{attribute 'no_assign'}
{attribute 'enable_dynamic_creation'}
{attribute 'no_explicit_call' := 'do not call this POU directly'}
FUNCTION_BLOCK FB_StringBuilder IMPLEMENTS I_StringBuilder, I_Enumerable
VAR CONSTANT
	Default_Capacity : T_Size := 256;
END_VAR
VAR
	{attribute 'hide'} 
	_Capacity : T_Size := THIS^.Default_Capacity;
	{attribute 'hide'} 
	_Length : T_Size := 0;
	_pBuffer : POINTER TO STRING := THIS^.Malloc(THIS^.Capacity);
END_VAR
VAR CONSTANT
	{attribute 'hide'} 
	_fbFree : FB_Free(THIS^._pBuffer) := ();
END_VAR

// Appends the given string to the end of the string builder's contents.
METHOD Append : I_StringBuilder
VAR_INPUT
	sValue : T_LongString;
END_VAR
Append := THIS^.AppendAny(sValue);
END_METHOD

// Appends the given value to the end of the string builder's contents.
METHOD AppendAny : I_StringBuilder
VAR_INPUT
	Value : ANY;
END_VAR
VAR
	bMalloced : BOOL := TRUE;
	Str_Len : T_Size;
	pValue : POINTER TO STRING;
END_VAR
AppendAny := THIS^;
CASE Value.TypeClass OF
	__SYSTEM.TYPE_CLASS.TYPE_STRING: 
		Str_Len := F_StrLen(Value.pValue);
		pValue := Value.pValue;
		bMalloced := FALSE;
		
	__SYSTEM.TYPE_CLASS.TYPE_WSTRING:
		Str_Len := TO_DINT(Tc2_Utilities.WLEN2(Value.pValue));
		pValue := THIS^.Malloc(Str_Len);
		Tc2_Utilities.WSTRING_TO_STRING2(pValue, Value.pValue, TO_UDINT(Str_Len));
		
	__SYSTEM.TYPE_CLASS.TYPE_BOOL,
	__SYSTEM.TYPE_CLASS.TYPE_BYTE,
	__SYSTEM.TYPE_CLASS.TYPE_WORD,
	__SYSTEM.TYPE_CLASS.TYPE_DWORD,
	__SYSTEM.TYPE_CLASS.TYPE_LWORD,
	__SYSTEM.TYPE_CLASS.TYPE_SINT,
	__SYSTEM.TYPE_CLASS.TYPE_INT,
	__SYSTEM.TYPE_CLASS.TYPE_DINT,
	__SYSTEM.TYPE_CLASS.TYPE_LINT,
	__SYSTEM.TYPE_CLASS.TYPE_USINT,
	__SYSTEM.TYPE_CLASS.TYPE_UINT,
	__SYSTEM.TYPE_CLASS.TYPE_UDINT,
	__SYSTEM.TYPE_CLASS.TYPE_ULINT,
	__SYSTEM.TYPE_CLASS.TYPE_REAL,
	__SYSTEM.TYPE_CLASS.TYPE_LREAL,
	__SYSTEM.TYPE_CLASS.TYPE_TIME,
	__SYSTEM.TYPE_CLASS.TYPE_LTIME,
	__SYSTEM.TYPE_CLASS.TYPE_DATE,
	__SYSTEM.TYPE_CLASS.TYPE_DATEANDTIME,
	__SYSTEM.TYPE_CLASS.TYPE_TIMEOFDAY,
	__SYSTEM.TYPE_CLASS.TYPE_POINTER:
		pValue := THIS^.Malloc(SIZEOF(T_LongString));
		pValue^ := F_AnyToString(Value);
		Str_Len := F_StrLen(pValue);
ELSE
	RETURN;
END_CASE

IF (THIS^.Length + Str_Len) >= THIS^.Capacity THEN
	THIS^.Reserve((THIS^.Length + Str_Len + 1)*2);
	END_IF

THIS^.Length := THIS^.Length + Str_Len;
F_StrLCat(THIS^._pBuffer, pValue, THIS^.Length + 1);

IF bMalloced THEN __DELETE(pValue); END_IF
END_METHOD

// !!!UNSAFE!!! THIS WILL APPEND UP TO THE NULL CHARACTER. IF NO NULL EXISTS, THIS WILL RUN FOREVER!
// | Append raw values directly to the internal string buffer. This is meant for appending dynamic strings to the string builder.
METHOD AppendBuffer : I_StringBuilder
VAR_INPUT
	pBuffer : POINTER TO BYTE;
END_VAR
VAR
	Str_Len : T_Size;
END_VAR
AppendBuffer := THIS^;
IF pBuffer = 0 THEN RETURN; END_IF
Str_Len := F_StrLen(pBuffer);

IF (THIS^.Length + Str_Len) >= THIS^.Capacity THEN
	THIS^.Reserve((THIS^.Length + Str_Len + 1)*2);
	END_IF
	
THIS^.Length := THIS^.Length + Str_Len;
F_StrLCat(THIS^._pBuffer, pBuffer, THIS^.Length + 1);
END_METHOD

// Appends a new line (\r\n or $r$n) to string builder's contents.
METHOD AppendLine : I_StringBuilder
AppendLine := THIS^;
THIS^.Append('$r$n');
END_METHOD

// Removes all ASCII white space (spaces, tabs, carriage returns, and linefeeds) from the beginning and end of string in the string builder
METHOD BTrim : I_StringBuilder
VAR
	Start, End, Length : T_Size := 0;
END_VAR
BTrim := THIS^;
IF THIS^.Length = 0 THEN RETURN; END_IF
End := THIS^.Length - 1;

WHILE ((Start <= End) AND THIS^.Is_Space(THIS^._pBuffer^[Start])) DO Start := Start  + 1; END_WHILE
WHILE ((End >= Start) AND THIS^.Is_Space(THIS^._pBuffer^[End])) DO End := End  - 1; END_WHILE

Length := end - start + 1;
F_MemMove(THIS^._pBuffer, ADR(THIS^._pBuffer^[Start]), Length);
THIS^.Length := Length;
THIS^._pBuffer^[THIS^.Length] := 0;
END_METHOD

// Number of bytes allocated in memory for the string builder's contents.
PROPERTY Capacity : T_Size
GET
Capacity := THIS^._Capacity;
END_GET
SET // PROTECTED
THIS^._Capacity := Capacity;
END_SET
END_PROPERTY

// Empties the string builder's contents, resetting its length to zero.
METHOD Clear : I_StringBuilder
Clear := THIS^;
THIS^.Free();
THIS^.Capacity := THIS^.Default_Capacity;
THIS^.Length := 0;
THIS^._pBuffer := THIS^.Malloc(THIS^.Capacity);
THIS^._pBuffer^[0] := 0;
END_METHOD

// Copies a subset of characters in the string builder from specified position at specified length to a string
METHOD CopySubstringTo : I_StringBuilder
VAR_INPUT
	Position, Length : T_Size;
	Value : ANY;
END_VAR
VAR
	pTemp : POINTER TO BYTE;
	pwsTemp : POINTER TO WSTRING;
END_VAR
CopySubstringTo := THIS^;
IF Value.pValue = 0 THEN RETURN; END_IF
CASE Value.TypeClass OF
	__SYSTEM.TYPE_CLASS.TYPE_STRING:
		Length := MIN(Length, Value.diSize - 1);
		IF (Position > THIS^.Length) OR_ELSE (Length <= 0) OR_ELSE (THIS^.Length = 0) THEN Value.pValue[0] := 0; RETURN; END_IF
		F_StrLCpy(Value.pValue, ADR(THIS^._pBuffer^[Position]), Length + 1);
		
	__SYSTEM.TYPE_CLASS.TYPE_WSTRING:
		Length := MIN(Length, (Value.diSize/2) - 1 );
		IF (Position > THIS^.Length) OR_ELSE (Length = 0) OR_ELSE (THIS^.Length = 0) THEN pwsTemp := Value.pValue; pwsTemp^ := ""; RETURN; END_IF
		pTemp := THIS^.Malloc(Length + 1);
		F_StrLCpy(pTemp, ADR(THIS^._pBuffer^[Position]), Length + 1);
		Tc2_Utilities.STRING_TO_WSTRING2(Value.pValue, pTemp, TO_UDINT((Length*2)+1));
		__DELETE(pTemp);
ELSE
	F_StrToAny(Value, THIS^.GetSubstring(Position, Length));
END_CASE
END_METHOD

// Copies contents of string builder to given string of any size
METHOD CopyTo : I_StringBuilder
VAR_INPUT
	Value : ANY;
END_VAR
CopyTo := THIS^;
IF THIS^._pBuffer = 0 THEN Value.pValue[0] := 0; RETURN; END_IF 
CASE Value.TypeClass OF
	__SYSTEM.TYPE_CLASS.TYPE_STRING:
		F_StrLCpy(Value.pValue, THIS^._pBuffer, Value.diSize);
	__SYSTEM.TYPE_CLASS.TYPE_WSTRING:
		Tc2_Utilities.STRING_TO_WSTRING2(Value.pValue, THIS^._pBuffer, TO_UDINT(Value.diSize));
ELSE
	F_StrToAny(Value, THIS^.GetString());
END_CASE
END_METHOD

// Dealloocates String from memory
METHOD PROTECTED Free
VAR_INPUT
END_VAR
IF THIS^._pBuffer <> 0 THEN __DELETE(THIS^._pBuffer); END_IF
THIS^.Capacity := 0;
END_METHOD

// !!!UNSAFE!!! DON'T FORGET TO RELEASE/DELETE FROM	MEMORY WHEN DONE!
// | Get a copy of the internal string buffer at the size of the string length + 1.
METHOD GetBuffer : I_StringBuilder
VAR_IN_OUT
	pBuffer : POINTER TO BYTE;
END_VAR
GetBuffer := THIS^;
pBuffer := THIS^.Malloc(THIS^.Length + 1);
F_StrLCpy(pBuffer, THIS^._pBuffer, THIS^.Length + 1);
END_METHOD

// Retrieves the number of bytes allocated in memory for the string builder's contents.
METHOD GetCapacity : I_StringBuilder
VAR_OUTPUT
	Capacity : T_Size;
END_VAR
GetCapacity := THIS^;
Capacity := THIS^.Capacity;
END_METHOD

// Gets character at specified position in the string builder
METHOD GetChar : T_Char
VAR_INPUT
	Position : T_Size;
END_VAR
IF Position < 0 THEN RETURN; END_IF
IF Position > THIS^.Length THEN RETURN; END_IF
GetChar[0] := THIS^._pBuffer^[Position];
END_METHOD

METHOD GetEnumerator : I_Enumerator
VAR_INST
	fbEnumerator : FB_StringBuilderEnumerator(THIS^);
END_VAR
GetEnumerator := fbEnumerator;
END_METHOD

// Retrieves the current size of string builder contents
METHOD GetLength : I_StringBuilder
VAR_OUTPUT
	Length : T_Size;
END_VAR
GetLength := THIS^;
Length := THIS^.Length;
END_METHOD

// Converts contents of string builder to string and returns them
METHOD GetString : T_LongString
THIS^.CopyTo(GetString);
END_METHOD

// Get a subset of characters in the string builder from specified position at specified length and returns them as a string
METHOD GetSubstring : T_LongString
VAR_INPUT
	Position, Length : T_Size;
END_VAR
THIS^.CopySubstringTo(Position, Length, GetSubstring);
END_METHOD

// Inserts the given string at the specified position.
METHOD Insert : I_StringBuilder
VAR_INPUT
	Position : T_Size;
	sValue : T_LongString;
END_VAR
Insert := THIS^.InsertAny(Position, sValue);
END_METHOD

// Inserts the given value at the specified position.
METHOD InsertAny : I_StringBuilder
VAR_INPUT
	Position : T_Size;
	Value : ANY;
END_VAR
VAR
	bMalloced : BOOL := TRUE;
	Str_Len : T_Size;
	pValue : POINTER TO STRING;
END_VAR
InsertAny := THIS^;
IF Position < 0 OR Position > THIS^.Length THEN RETURN; END_IF 
CASE Value.TypeClass OF
	__SYSTEM.TYPE_CLASS.TYPE_STRING: 
		Str_Len := F_StrLen(Value.pValue);
		pValue := Value.pValue;
		bMalloced := FALSE;
	
	__SYSTEM.TYPE_CLASS.TYPE_WSTRING:
		Str_Len := TO_DINT(Tc2_Utilities.WLEN2(Value.pValue));
		pValue := THIS^.Malloc(Str_Len);
		Tc2_Utilities.WSTRING_TO_STRING2(pValue, Value.pValue, TO_UDINT(Str_Len));

	__SYSTEM.TYPE_CLASS.TYPE_BOOL,
	__SYSTEM.TYPE_CLASS.TYPE_BYTE,
	__SYSTEM.TYPE_CLASS.TYPE_WORD,
	__SYSTEM.TYPE_CLASS.TYPE_DWORD,
	__SYSTEM.TYPE_CLASS.TYPE_LWORD,
	__SYSTEM.TYPE_CLASS.TYPE_SINT,
	__SYSTEM.TYPE_CLASS.TYPE_INT,
	__SYSTEM.TYPE_CLASS.TYPE_DINT,
	__SYSTEM.TYPE_CLASS.TYPE_LINT,
	__SYSTEM.TYPE_CLASS.TYPE_USINT,
	__SYSTEM.TYPE_CLASS.TYPE_UINT,
	__SYSTEM.TYPE_CLASS.TYPE_UDINT,
	__SYSTEM.TYPE_CLASS.TYPE_ULINT,
	__SYSTEM.TYPE_CLASS.TYPE_REAL,
	__SYSTEM.TYPE_CLASS.TYPE_LREAL,
	__SYSTEM.TYPE_CLASS.TYPE_TIME,
	__SYSTEM.TYPE_CLASS.TYPE_LTIME,
	__SYSTEM.TYPE_CLASS.TYPE_DATE,
	__SYSTEM.TYPE_CLASS.TYPE_DATEANDTIME,
	__SYSTEM.TYPE_CLASS.TYPE_TIMEOFDAY,
	__SYSTEM.TYPE_CLASS.TYPE_POINTER:
		pValue := THIS^.Malloc(SIZEOF(T_LongString));
		pValue^ := F_AnyToString(Value);
		Str_Len := F_StrLen(pValue);
ELSE
	RETURN;
END_CASE

IF (THIS^.Length + Str_Len) >= THIS^.Capacity THEN
	THIS^.Reserve((THIS^.Length + Str_Len + 1)*2);
	END_IF

F_MemMove(THIS^._pBuffer + TO_UDINT(Position) + TO_UDINT(Str_Len), THIS^._pBuffer + TO_UDINT(Position), THIS^.Length - Position + 1);
F_MemCpy(THIS^._pBuffer + TO_UDINT(Position), pValue, Str_Len); 
THIS^.Length := THIS^.Length + Str_Len;

IF bMalloced THEN __DELETE(pValue); END_IF
END_METHOD

// !!!UNSAFE!!! THIS WILL INSERT UP TO THE NULL CHARACTER. IF NO NULL EXISTS, THIS WILL RUN FOREVER!
// | Inserts raw values directly to the internal string buffer at the specified position. This is meant for inserting dynamic strings to the string builder.
METHOD InsertBuffer : I_StringBuilder
VAR_INPUT
	Position : T_Size;
	pBuffer : POINTER TO BYTE;
END_VAR
VAR
	Str_Len : T_Size;
END_VAR
InsertBuffer := THIS^;
IF pBuffer = 0 OR Position < 0 OR Position > THIS^.Length THEN RETURN; END_IF
Str_Len := F_StrLen(pBuffer);

IF (THIS^.Length + Str_Len) >= THIS^.Capacity THEN
	THIS^.Reserve((THIS^.Length + Str_Len + 1)*2);
	END_IF

F_MemMove(THIS^._pBuffer + TO_UDINT(Position) + TO_UDINT(Str_Len), THIS^._pBuffer + TO_UDINT(Position), THIS^.Length - Position + 1);
F_MemCpy(THIS^._pBuffer + TO_UDINT(Position), pBuffer, Str_Len); 
THIS^.Length := THIS^.Length + Str_Len;
END_METHOD

METHOD PROTECTED Is_Space : BOOL
VAR_INPUT
	nChar : BYTE;
END_VAR
Is_Space := (nChar = 32) OR_ELSE (nChar = 9) OR_ELSE (nChar = 10) OR_ELSE (nChar = 13) OR_ELSE (nChar = 12) OR_ELSE (nChar = 11);
END_METHOD

// Joins/Merges the string contents of the current string builder with that on the specified string builder at the specified position
METHOD Join : I_StringBuilder
VAR_INPUT
	Position : T_Size;
	ipString_Builder : I_StringBuilder;
END_VAR
VAR
	pTemp : POINTER TO BYTE;
END_VAR
Join := THIS^;
IF ipString_Builder = 0 THEN RETURN; END_IF
ipString_Builder.GetBuffer(pTemp);
THIS^.InsertBuffer(Position, pTemp);
CASE Tc2_System.F_CheckMemoryArea(pTemp, 1) OF 
	E_TcMemoryArea.Dynamic: __DELETE(pTemp);
END_CASE
END_METHOD

// Current size of string builder contents
PROPERTY Length : T_Size
GET
VAR
	i : UDINT;
END_VAR
Length := THIS^._Length;
END_GET
SET // PROTECTED
THIS^._Length := Length;
END_SET
END_PROPERTY

// Removes all ASCII white space (spaces, tabs, carriage returns, and linefeeds) from the beginning of string in the string builder
METHOD LTrim : I_StringBuilder
VAR
	Start, End, Length : T_Size := 0;
END_VAR
LTrim := THIS^;
IF THIS^.Length = 0 THEN RETURN; END_IF
End := THIS^.Length - 1;

WHILE ((Start <= End) AND THIS^.Is_Space(THIS^._pBuffer^[Start])) DO Start := Start + 1; END_WHILE

Length := end - start + 1;
F_MemMove(THIS^._pBuffer, ADR(THIS^._pBuffer^[Start]), Length);
THIS^.Length := Length;
THIS^._pBuffer^[THIS^.Length] := 0;
END_METHOD

// Allocates memory on the heap for a string of defined size
METHOD PROTECTED Malloc : POINTER TO STRING
VAR_INPUT
	Size : T_Size;
END_VAR
Malloc := __NEW(BYTE, TO_UDINT(Size));
END_METHOD

// Removes the characters in the string builder from specified position at specified length.+
METHOD Remove : I_StringBuilder
VAR_INPUT
	Position, Length : T_Size;
END_VAR
Remove := THIS^;
IF Position + Length > THIS^.Length OR Position < 0 OR Length <= 0 OR Position > THIS^.Length THEN RETURN; END_IF
F_MemMove(ADR(THIS^._pBuffer^[Position]), ADR(THIS^._pBuffer^[Position + Length]), THIS^.Length - (Position + Length) + 1);
THIS^.Length := THIS^.Length - Length;
END_METHOD

// Replaces the instance of the old string in the string builder with the new string.
// If bReplace_All = TRUE, all instances of the old string are placed, else only the first instance.
METHOD Replace : I_StringBuilder
VAR_INPUT
	sOld_Value,
	sNew_Value : T_LongString;
	bReplace_All : BOOL;
END_VAR
Replace := THIS^.ReplaceAny(sOld_Value,sNew_Value, bReplace_All);
END_METHOD

// Replaces the instance of the old value in the string builder with the new value.
// If bReplace_All = TRUE, all instances of the old value are placed, else only the first instance.
METHOD ReplaceAny : I_StringBuilder
VAR_INPUT
	Old_Value : ANY;
	New_Value : ANY;
	bReplace_All : BOOL;
END_VAR
VAR
	Position, 
	Old_Str_Len,
	New_Str_len : T_Size;
END_VAR
ReplaceAny := THIS^;
IF NOT(F_IsAnyToStringCompatable(Old_Value)) OR_ELSE NOT(F_IsAnyToStringCompatable(New_Value)) THEN RETURN; END_IF

Old_Str_Len := F_AnyStringLength(Old_Value);
New_Str_Len := F_AnyStringLength(New_Value);

WHILE Position < THIS^.Length DO
	THIS^.SearchAny(Old_Value, Position, Position => Position);
	THIS^.Remove(Position, Old_Str_Len);
	THIS^.InsertAny(Position, New_Value);
	IF NOT bReplace_All OR Position < 0 THEN EXIT; END_IF
	Position := Position + New_Str_Len;
	END_WHILE
END_METHOD

METHOD PROTECTED Reserve
VAR_INPUT
	Capacity : T_Size;
END_VAR
VAR
	pTemp : POINTER TO STRING;
END_VAR
IF Capacity <= THIS^.Capacity THEN RETURN; END_IF
pTemp := THIS^.Malloc(Capacity);
F_StrLCpy(pTemp, THIS^._pBuffer, Capacity);
THIS^.Free();
THIS^._pBuffer := pTemp;
THIS^.Capacity := Capacity;
END_METHOD

// Reverses the string contents in the string builder
METHOD Reverse : I_StringBuilder
VAR
	i : T_Size;
	nTemp : BYTE;
END_VAR
Reverse := THIS^;
IF THIS^.Length <= 0 THEN RETURN; END_IF
FOR i := 0 TO (THIS^.Length/2)-1 DO
	nTemp := THIS^._pBuffer^[i];
	THIS^._pBuffer^[i] := THIS^._pBuffer^[THIS^.Length - i - 1];
	THIS^._pBuffer^[THIS^.Length - i - 1] := nTemp;
	END_FOR
END_METHOD

// Removes all ASCII white space (spaces, tabs, carriage returns, and linefeeds) from the end of string in the string builder
METHOD RTrim : I_StringBuilder
VAR
	Start, End, Length : T_Size := 0;
END_VAR
RTrim := THIS^;
IF THIS^.Length = 0 THEN RETURN; END_IF
End := THIS^.Length - 1;

WHILE ((End >= Start) AND THIS^.Is_Space(THIS^._pBuffer^[End])) DO End := End  - 1; END_WHILE

Length := end - start + 1;
F_MemMove(THIS^._pBuffer, ADR(THIS^._pBuffer^[Start]), Length);
THIS^.Length := Length;
THIS^._pBuffer^[THIS^.Length] := 0;
END_METHOD

// Finds the position of the first instance of a given string in the content's of the string builder from a starting position
METHOD Search : I_StringBuilder
VAR_INPUT
	sValue : T_LongString;
	Start_Position : T_Size;
END_VAR
VAR_OUTPUT
	Position : T_Size;
END_VAR
Search := THIS^.SearchAny(sValue,Start_Position, Position => Position);
END_METHOD

// Finds the position of the first instance of a given value in the content's of the string builder from a starting position
METHOD SearchAny : I_StringBuilder
VAR_INPUT
	Value : ANY;
	Start_Position : T_Size;
END_VAR
VAR_OUTPUT
	Position : T_Size := -1;
END_VAR
VAR
	bMalloced : BOOL := TRUE;
	Str_Len : T_Size;
	pValue, pLoc : POINTER TO STRING;
END_VAR
SearchAny := THIS^;
IF Start_Position < 0 OR Start_Position > THIS^.Length - 1 THEN RETURN; END_IF
CASE Value.TypeClass OF
	__SYSTEM.TYPE_CLASS.TYPE_STRING: 
		pValue := Value.pValue;
		bMalloced := FALSE;
		
	__SYSTEM.TYPE_CLASS.TYPE_WSTRING:
		Str_Len := TO_DINT(Tc2_Utilities.WLEN2(Value.pValue));
		pValue := THIS^.Malloc(Str_Len + 1);
		Tc2_Utilities.WSTRING_TO_STRING2(pValue, Value.pValue, TO_UDINT(Str_Len));
		
	__SYSTEM.TYPE_CLASS.TYPE_BOOL,
	__SYSTEM.TYPE_CLASS.TYPE_BYTE,
	__SYSTEM.TYPE_CLASS.TYPE_WORD,
	__SYSTEM.TYPE_CLASS.TYPE_DWORD,
	__SYSTEM.TYPE_CLASS.TYPE_LWORD,
	__SYSTEM.TYPE_CLASS.TYPE_SINT,
	__SYSTEM.TYPE_CLASS.TYPE_INT,
	__SYSTEM.TYPE_CLASS.TYPE_DINT,
	__SYSTEM.TYPE_CLASS.TYPE_LINT,
	__SYSTEM.TYPE_CLASS.TYPE_USINT,
	__SYSTEM.TYPE_CLASS.TYPE_UINT,
	__SYSTEM.TYPE_CLASS.TYPE_UDINT,
	__SYSTEM.TYPE_CLASS.TYPE_ULINT,
	__SYSTEM.TYPE_CLASS.TYPE_REAL,
	__SYSTEM.TYPE_CLASS.TYPE_LREAL,
	__SYSTEM.TYPE_CLASS.TYPE_TIME,
	__SYSTEM.TYPE_CLASS.TYPE_LTIME,
	__SYSTEM.TYPE_CLASS.TYPE_DATE,
	__SYSTEM.TYPE_CLASS.TYPE_DATEANDTIME,
	__SYSTEM.TYPE_CLASS.TYPE_TIMEOFDAY,
	__SYSTEM.TYPE_CLASS.TYPE_POINTER:
		pValue := THIS^.Malloc(SIZEOF(T_LongString));
		pValue^ := F_AnyToString(Value);
ELSE
	RETURN;
END_CASE
pLoc := F_StrStr(ADR(THIS^._pBuffer^[Start_Position]), pValue);
IF bMalloced THEN __DELETE(pValue); END_IF
IF pLoc = 0 THEN RETURN; END_IF
Position := TO_DINT(pLoc - THIS^._pBuffer);
END_METHOD

// Appends selected characters from the current string builder to the selected string builder
METHOD Split : I_StringBuilder
VAR_INPUT
	Position, Length : T_Size;
	ipStringBuilder : I_StringBuilder;
END_VAR
VAR
	Char : T_Char;
	i, End_Position : T_Size;
END_VAR
Split := THIS^;
IF ipStringBuilder = 0 THEN RETURN; END_IF
IF (Position > THIS^.Length) OR_ELSE (Length <= 0) OR_ELSE (THIS^.Length = 0) THEN RETURN; END_IF
End_Position := Position + Length;
IF End_Position > THIS^.Length THEN End_Position := THIS^.Length; END_IF

FOR i := Position TO End_Position - 1 DO
	Char[0] := THIS^._pBuffer^[i];
	ipStringBuilder.Append(Char);
	END_FOR
END_METHOD

// Reduces the capacity of the string builder to match the size of its contents, potentially reducing memory usage.
METHOD StrinkToFit : I_StringBuilder
VAR
	pTemp : POINTER TO STRING;
END_VAR
StrinkToFit := THIS^;
IF THIS^.Capacity > (THIS^.Length + 1) THEN
	pTemp := THIS^.Malloc(THIS^.Length + 1);
	F_StrLCpy(pTemp, THIS^._pBuffer, THIS^.Length + 1);
	THIS^.Free();
	THIS^._pBuffer := pTemp;
	THIS^.Capacity := THIS^.Length + 1;
	END_IF
END_METHOD

// Converts all alphabetic characters in string builder to lowercase characters
METHOD ToLowercase : I_StringBuilder
VAR
	i : T_Size;
END_VAR
ToLowercase := THIS^;
IF THIS^.Length = 0 THEN RETURN; END_IF
FOR i := 0 TO THIS^.Length - 1 DO 
	IF THIS^._pBuffer^[i] >= 65 AND THIS^._pBuffer^[i]<= 90 THEN 
		THIS^._pBuffer^[i] := THIS^._pBuffer^[i] + 32; 
		END_IF
	END_FOR
END_METHOD

// Converts all alphabetic characters in string builder to uppercase characters
METHOD ToUppercase : I_StringBuilder
VAR
	i : T_Size;
END_VAR
ToUppercase := THIS^;
IF THIS^.Length = 0 THEN RETURN; END_IF
FOR i := 0 TO THIS^.Length - 1 DO 
	IF THIS^._pBuffer^[i] >= 97 AND THIS^._pBuffer^[i]<= 122 THEN 
		THIS^._pBuffer^[i] := THIS^._pBuffer^[i] - 32; 
		END_IF
	END_FOR
END_METHOD

END_FUNCTION_BLOCK

(* stored: Version 1.1.0.1, ProductVersion 3.1.4024.4
   POU FB_StringBuilder: Id {4bfd7369-678a-4946-9112-ed6456534c78}, SpecialFunc None
   Folder Private: Id {3c3e121d-c945-45bd-b6bd-25e0688a969f}
   Folder Protected: Id {4477869e-92c9-4a27-9c5f-70db177e2987}
   Method Append: Id {01d06d20-00ca-4ddb-ac88-d57d11106c30}
   Method AppendAny: Id {bbc36120-bb82-4698-869d-56f829e1ec49}
   Method AppendBuffer: Id {ab096c91-db1d-45c9-9802-c30c8edda13d}
   Method AppendLine: Id {47bb1f01-ff10-4f2d-b428-52f8d3d2a7d9}
   Method BTrim: Id {baabad4b-9105-41bd-a958-cfa16de0468c}
   Property Capacity: Id {7a1eab10-ae41-45cb-bda3-567ca6b8ca2b}
   Get Get: Id {737e6d02-df74-49cc-8ebb-4ee9bfcdb284}
   Set Set: Id {bd69bbff-5cad-44c9-9d07-120ef29a443c}
   Method Clear: Id {783fdd2d-09f4-4c32-a081-6c3bbdd1c93b}
   Method CopySubstringTo: Id {f5cac2bf-671f-41eb-b88a-0fca63f88e19}
   Method CopyTo: Id {6dee6299-607f-420c-87bf-d6ba465e5957}
   Method Free: Id {f566a732-3ec5-4648-b07b-3c7c9489a31b}
   Method GetBuffer: Id {2c0611a8-2ab7-47c6-a25b-f84c5611fd08}
   Method GetCapacity: Id {3f0a7335-54fd-4d8c-93df-4a361b67bb88}
   Method GetChar: Id {de5c8ed1-c067-4d7b-922b-537b0e46a5f7}
   Method GetEnumerator: Id {88dbe339-378c-45d6-bb2a-ab340943596d}
   Method GetLength: Id {28151eb1-85c5-450d-9b23-ac2e54cd2b0d}
   Method GetString: Id {60b5f273-83ef-4a38-98c6-d4a9815f983f}
   Method GetSubstring: Id {b9f92418-c277-4297-84a9-e70a422ab510}
   Method Insert: Id {0f715bee-e923-4cb0-9c9d-189ede2e8e1b}
   Method InsertAny: Id {108fe9a3-24cb-4e3e-a1c9-a5948a95313d}
   Method InsertBuffer: Id {e4fce2fa-3e69-42b4-8422-9b4b1cd1d44e}
   Method Is_Space: Id {1b805b4e-1581-4fd2-adcb-7bfeeedf6485}
   Method Join: Id {9dc96dcf-9c4f-4a3b-8f16-54ac73d078a5}
   Property Length: Id {42ee92eb-6db1-44ae-878f-3eb5c5f39c6c}
   Get Get: Id {fe15fef6-4a27-449f-8986-a39081f27e7c}
   Set Set: Id {7731a0b4-0ff8-414a-a7ad-09cc142375d9}
   Method LTrim: Id {4df3ac1a-8e0e-4e50-b32f-ac510ccc12c1}
   Method Malloc: Id {a88316a6-1528-4842-9841-0f6d45c046b9}
   Method Remove: Id {76f04ac2-7427-4649-af11-5e4b326e4f67}
   Method Replace: Id {319dcc88-3e0c-48b4-bf59-3a020c9b84cb}
   Method ReplaceAny: Id {3a55c232-be68-40d3-aae3-79b945f2fdb3}
   Method Reserve: Id {20490fb2-0dc3-481b-b6b6-14608ad46bd6}
   Method Reverse: Id {230c981c-7bc4-4cc1-81a8-f260fa2c7145}
   Method RTrim: Id {0abf2bf8-662e-4545-9933-322af8689797}
   Method Search: Id {38591f35-eb58-43a1-803d-68119051cbc2}
   Method SearchAny: Id {ab6ebf17-ea26-4de6-8473-c7633d94ec15}
   Method Split: Id {4a618ce1-9fc5-46aa-bd25-d7a2c05a8ab9}
   Method StrinkToFit: Id {0335a2b7-1853-42a3-854f-56422bd5149a}
   Method ToLowercase: Id {a1fcd3aa-8fa4-4184-b06b-5118ba2c163f}
   Method ToUppercase: Id {bf56b332-7403-4ffc-afda-d2a8ff11b9af} *)
